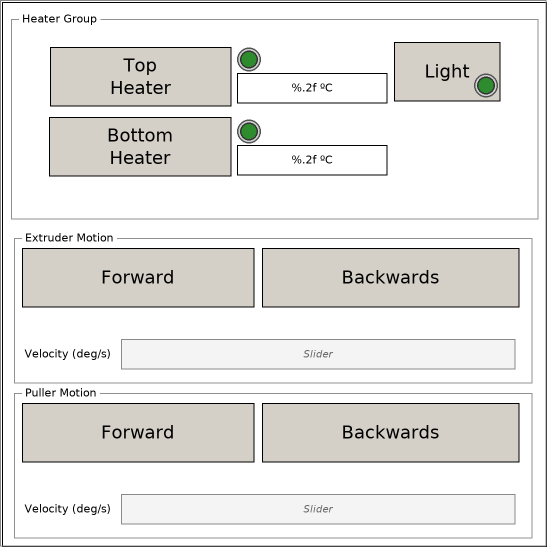
VISUALIZATION ManualHMI  // 547x547
    Rectangle (2,2 545x545)
    GroupBox (11,11 527x208), "Heater Group"
        Rectangle (39,36 181x59), "Top Heater"
            toggle HMI.Bt_ManHeatTop
        Rectangle (226,62 150x30), "%.2f ºC", text variable: GVL.TempTerT
        Rectangle (226,134 150x30), "%.2f ºC", text variable: GVL.TempTerB
        Lamp1 (224,107 28x27), variable: IO.Q_HeaterB, style: Lamp-Lamp1-Green
        Lamp1 (224,35 28x27), variable: IO.Q_HeaterT, style: Lamp-Lamp1-Green
        Rectangle (38,106 182x59), "Bottom Heater"
            toggle HMI.Bt_ManHeatBot
        Rectangle (383,31 106x59), "Light"
            toggle HMI.Bt_Light
        Lamp1 (461,61 28x27), variable: IO.Q_VisionLight, style: Lamp-Lamp1-Green
    GroupBox (14,230 518x153), "Extruder Motion"
        Rectangle (8,18 232x59), "Forward"
            tap HMI.Bt_ManForwardExtruder
        Rectangle (248,18 257x59), "Backwards"
            tap HMI.Bt_ManBackwardsExtruder
        Slider (107,109 394x30), variable: HMI.Tb_ManVelExtruder, scale 0..720
        Label (2,109 104x30), "Velocity (deg/s)"
    GroupBox (14,385 518x153), "Puller Motion"
        Rectangle (8,18 232x59), "Forward"
            tap HMI.Bt_ManForwardPuller
        Rectangle (248,18 257x59), "Backwards"
            tap HMI.Bt_ManBackwardsPuller
        Slider (107,109 394x30), variable: HMI.Tb_ManVelPuller, scale 0..720
        Label (2,109 104x30), "Velocity (deg/s)"
END_VISUALIZATION

(* stored: Version 1.1.0.1, ProductVersion 3.1.4024.9
   Visu ManualHMI: Id {239d5e59-9cf8-44cf-b394-bf771424e551} *)
